DECL FDAT FP87={TOOL_NO 1,BASE_NO 0,IPO_FRAME #BASE,POINT2[] " ",TQ_STATE FALSE}
DECL PDAT PPDAT66={ACC 100.000,APO_DIST 100.000,APO_MODE #CPTP,GEAR_JERK 50.0000}
DECL E6POS XP87={X 1397.26331,Y -207.500198,Z 1611.62207,A -136.868607,B 85.8667068,C -39.2035751,S 2,T 2,E1 229.997360,E2 195.002197,E3 195.004211,E4 0.0,E5 0.0,E6 0.0}
DECL ATBg_Crater_T AC_WDAT46={JobModeId -187662529,ParamSetId -1375177600,CraterTime 0.100000,PostflowTime 0.100000,Channel1 30.0000,Channel2 1.00000,Channel3 0.0,Channel4 0.0,Channel5 0.0,Channel6 0.0,Channel7 0.0,Channel8 0.0,BurnBackTime 0.0}
DECL FDAT FP88={TOOL_NO 1,BASE_NO 0,IPO_FRAME #BASE,POINT2[] " ",TQ_STATE FALSE}
DECL LDAT LCPDAT25={ACC 100.000,APO_DIST 100.000,APO_FAC 50.0000,AXIS_VEL 100.000,AXIS_ACC 100.000,ORI_TYP #VAR,CIRC_TYP #BASE,JERK_FAC 50.0000,GEAR_JERK 50.0000,EXAX_IGN 0}
DECL E6POS XP88={X 1397.26331,Y -207.500198,Z 1611.62207,A -136.868607,B 85.8667068,C -39.2035751,S 2,T 2,E1 229.997360,E2 195.002197,E3 195.004211,E4 0.0,E5 0.0,E6 0.0}
DECL E6POS XP89={X 1306.19275,Y -196.588913,Z 1703.97925,A -68.7830734,B 86.4150162,C 29.0020599,S 2,T 2,E1 229.997360,E2 195.002197,E3 195.004211,E4 0.0,E5 0.0,E6 0.0}
DECL FDAT FP89={TOOL_NO 1,BASE_NO 0,IPO_FRAME #BASE,POINT2[] " ",TQ_STATE FALSE}
DECL PDAT PPDAT67={VEL 100.000,ACC 100.000,APO_DIST 100.000,APO_MODE #CDIS,GEAR_JERK 50.0000,EXAX_IGN 3}
DECL ATBg_Start_T AS_WDAT47={JobModeId -187662529,ParamSetId 687014726,StartTime 0.0,PreFlowTime 0.100000,Channel1 30.0000,Channel2 1.00000,Channel3 0.0,Channel4 0.0,Channel5 0.0,Channel6 0.0,Channel7 0.0,Channel8 0.0,PurgeTime 0.0}
DECL ATBg_Weld_T AW_WDAT47={JobModeId -187662529,ParamSetId -430485013,Velocity 0.00830000,Channel1 30.0000,Channel2 1.00000,Channel3 0.0,Channel4 0.0,Channel5 0.0,Channel6 0.0,Channel7 0.0,Channel8 0.0}
DECL WTCg_WeaveDefinition_T WV_WDAT47={Pattern #None,Length 4.00000,Amplitude 2.00000,Angle 0.0}
DECL FDAT FP90={TOOL_NO 1,BASE_NO 0,IPO_FRAME #BASE,POINT2[] " ",TQ_STATE FALSE}
DECL PDAT PPDAT68={ACC 100.000,APO_DIST 100.000,APO_MODE #CPTP,GEAR_JERK 50.0000}
DECL E6POS XP90={X 1232.65955,Y -891.276917,Z 1635.28589,A -96.7124100,B 54.7162971,C 6.76454,S 2,T 10,E1 229.997360,E2 195.002197,E3 195.004211,E4 0.0,E5 0.0,E6 0.0}
DECL ATBg_Crater_T AC_WDAT48={JobModeId -187662529,ParamSetId -1375177600,CraterTime 0.100000,PostflowTime 0.100000,Channel1 30.0000,Channel2 1.00000,Channel3 0.0,Channel4 0.0,Channel5 0.0,Channel6 0.0,Channel7 0.0,Channel8 0.0,BurnBackTime 0.0}
DECL FDAT FP91={TOOL_NO 1,BASE_NO 0,IPO_FRAME #BASE,POINT2[] " ",TQ_STATE FALSE}
DECL LDAT LCPDAT26={ACC 100.000,APO_DIST 100.000,APO_FAC 50.0000,AXIS_VEL 100.000,AXIS_ACC 100.000,ORI_TYP #VAR,CIRC_TYP #BASE,JERK_FAC 50.0000,GEAR_JERK 50.0000,EXAX_IGN 0}
DECL E6POS XP91={X 1232.65955,Y -891.276917,Z 1635.28589,A -96.7124100,B 54.7162971,C 6.76454,S 2,T 10,E1 229.997360,E2 195.002197,E3 195.004211,E4 0.0,E5 0.0,E6 0.0}
DECL E6POS XP92={X 1054.34692,Y -757.859863,Z 1864.28418,A -84.9267426,B 47.8384056,C 21.8099632,S 2,T 10,E1 229.997360,E2 195.002197,E3 195.004211,E4 0.0,E5 0.0,E6 0.0}
DECL FDAT FP92={TOOL_NO 1,BASE_NO 0,IPO_FRAME #BASE,POINT2[] " ",TQ_STATE FALSE}
DECL PDAT PPDAT69={VEL 100.000,ACC 100.000,APO_DIST 100.000,APO_MODE #CDIS,GEAR_JERK 50.0000,EXAX_IGN 3}
DECL E6POS XP93={X 1192.32471,Y 472.459,Z 1776.73877,A 83.1334229,B 67.4761200,C 156.576218,S 2,T 35,E1 229.997406,E2 195.002228,E3 195.004227,E4 0.0,E5 0.0,E6 0.0}
DECL FDAT FP93={TOOL_NO 1,BASE_NO 0,IPO_FRAME #BASE,POINT2[] " ",TQ_STATE FALSE}
DECL PDAT PPDAT70={VEL 100.000,ACC 100.000,APO_DIST 100.000,APO_MODE #CDIS,GEAR_JERK 50.0000,EXAX_IGN 3}
DECL E6POS XP94={X 1203.56567,Y 245.655396,Z 1802.88013,A 72.3533630,B 68.4953918,C 154.352661,S 2,T 35,E1 229.997391,E2 195.002228,E3 195.004227,E4 0.0,E5 0.0,E6 0.0}
DECL FDAT FP94={TOOL_NO 1,BASE_NO 0,IPO_FRAME #BASE,POINT2[] " ",TQ_STATE FALSE}
DECL PDAT PPDAT71={VEL 100.000,ACC 100.000,APO_DIST 100.000,APO_MODE #CDIS,GEAR_JERK 50.0000,EXAX_IGN 3}
DECL E6POS XP95={X 1366.39880,Y 202.321213,Z 1652.72510,A 92.5657654,B 80.7616730,C 174.120758,S 2,T 35,E1 229.997360,E2 195.002197,E3 195.004211,E4 0.0,E5 0.0,E6 0.0}
DECL FDAT FP95={TOOL_NO 1,BASE_NO 0,IPO_FRAME #BASE,POINT2[] " ",TQ_STATE FALSE}
DECL PDAT PPDAT72={VEL 100.000,ACC 100.000,APO_DIST 100.000,APO_MODE #CDIS,GEAR_JERK 50.0000,EXAX_IGN 3}
DECL E6POS XP96={X 1171.60815,Y -889.236572,Z 1696.34497,A -96.0087738,B 50.3284950,C 9.56970692,S 2,T 10,E1 190.873,E2 195.002197,E3 195.004211,E4 0.0,E5 0.0,E6 0.0}
DECL FDAT FP96={TOOL_NO 1,BASE_NO 0,IPO_FRAME #BASE,POINT2[] " ",TQ_STATE FALSE}
DECL PDAT PPDAT73={VEL 100.000,ACC 100.000,APO_DIST 100.000,APO_MODE #CDIS,GEAR_JERK 50.0000,EXAX_IGN 3}
DECL ATBg_Start_T AS_WDAT49={JobModeId -187662529,ParamSetId 687014726,StartTime 0.0,PreFlowTime 0.100000,Channel1 30.0000,Channel2 1.00000,Channel3 0.0,Channel4 0.0,Channel5 0.0,Channel6 0.0,Channel7 0.0,Channel8 0.0,PurgeTime 0.0}
DECL ATBg_Weld_T AW_WDAT49={JobModeId -187662529,ParamSetId -430485013,Velocity 0.00830000,Channel1 30.0000,Channel2 1.00000,Channel3 0.0,Channel4 0.0,Channel5 0.0,Channel6 0.0,Channel7 0.0,Channel8 0.0}
DECL WTCg_WeaveDefinition_T WV_WDAT49={Pattern #None,Length 4.00000,Amplitude 2.00000,Angle 0.0}
DECL FDAT FP97={TOOL_NO 1,BASE_NO 0,IPO_FRAME #BASE,POINT2[] " ",TQ_STATE FALSE}
DECL PDAT PPDAT74={ACC 100.000,APO_DIST 100.000,APO_MODE #CPTP,GEAR_JERK 50.0000}
DECL E6POS XP97={X 1206.43689,Y -921.566711,Z 1635.16187,A -94.9919662,B 61.2246590,C 10.2442360,S 2,T 10,E1 190.873,E2 195.002197,E3 195.004211,E4 0.0,E5 0.0,E6 0.0}
DECL ATBg_Crater_T AC_WDAT50={JobModeId -187662529,ParamSetId -1375177600,CraterTime 0.100000,PostflowTime 0.100000,Channel1 30.0000,Channel2 1.00000,Channel3 0.0,Channel4 0.0,Channel5 0.0,Channel6 0.0,Channel7 0.0,Channel8 0.0,BurnBackTime 0.0}
DECL FDAT FP98={TOOL_NO 1,BASE_NO 0,IPO_FRAME #BASE,POINT2[] " ",TQ_STATE FALSE}
DECL LDAT LCPDAT27={ACC 100.000,APO_DIST 100.000,APO_FAC 50.0000,AXIS_VEL 100.000,AXIS_ACC 100.000,ORI_TYP #VAR,CIRC_TYP #BASE,JERK_FAC 50.0000,GEAR_JERK 50.0000,EXAX_IGN 0}
DECL E6POS XP98={X 1206.43689,Y -921.566711,Z 1635.16187,A -94.9919662,B 61.2246590,C 10.2442360,S 2,T 10,E1 190.873,E2 195.002197,E3 195.004211,E4 0.0,E5 0.0,E6 0.0}
DECL ATBg_Crater_T AC_WDAT51={JobModeId -187662529,ParamSetId -1375177600,CraterTime 0.100000,PostflowTime 0.100000,Channel1 30.0000,Channel2 1.00000,Channel3 0.0,Channel4 0.0,Channel5 0.0,Channel6 0.0,Channel7 0.0,Channel8 0.0,BurnBackTime 0.0}
DECL FDAT FP99={TOOL_NO 1,BASE_NO 0,IPO_FRAME #BASE,POINT2[] " ",TQ_STATE FALSE}
DECL LDAT LCPDAT28={ACC 100.000,APO_DIST 100.000,APO_FAC 50.0000,AXIS_VEL 100.000,AXIS_ACC 100.000,ORI_TYP #VAR,CIRC_TYP #BASE,JERK_FAC 50.0000,GEAR_JERK 50.0000,EXAX_IGN 0}
DECL E6POS XP99={X 1194.17407,Y -927.370056,Z 1636.72192,A -96.0782471,B 61.4487839,C 9.53255939,S 2,T 10,E1 190.873,E2 195.002197,E3 195.004211,E4 0.0,E5 0.0,E6 0.0}
DECL ATBg_Start_T AS_WDAT52={JobModeId -187662529,ParamSetId 687014726,StartTime 0.0,PreFlowTime 0.100000,Channel1 30.0000,Channel2 1.00000,Channel3 0.0,Channel4 0.0,Channel5 0.0,Channel6 0.0,Channel7 0.0,Channel8 0.0,PurgeTime 0.0}
DECL ATBg_Weld_T AW_WDAT52={JobModeId -187662529,ParamSetId -430485013,Velocity 0.00830000,Channel1 30.0000,Channel2 1.00000,Channel3 0.0,Channel4 0.0,Channel5 0.0,Channel6 0.0,Channel7 0.0,Channel8 0.0}
DECL WTCg_WeaveDefinition_T WV_WDAT52={Pattern #None,Length 4.00000,Amplitude 2.00000,Angle 0.0}
DECL FDAT FP100={TOOL_NO 1,BASE_NO 0,IPO_FRAME #BASE,POINT2[] " ",TQ_STATE FALSE}
DECL PDAT PPDAT75={ACC 100.000,APO_DIST 100.000,APO_MODE #CPTP,GEAR_JERK 50.0000}
DECL E6POS XP100={X 1254.47900,Y -806.532104,Z 1613.77075,A -96.0353394,B 70.1869659,C 2.27105737,S 2,T 10,E1 190.873,E2 195.002197,E3 195.004211,E4 0.0,E5 0.0,E6 0.0}
DECL ATBg_Crater_T AC_WDAT53={JobModeId -187662529,ParamSetId -1375177600,CraterTime 0.100000,PostflowTime 0.100000,Channel1 30.0000,Channel2 1.00000,Channel3 0.0,Channel4 0.0,Channel5 0.0,Channel6 0.0,Channel7 0.0,Channel8 0.0,BurnBackTime 0.0}
DECL FDAT FP101={TOOL_NO 1,BASE_NO 0,IPO_FRAME #BASE,POINT2[] " ",TQ_STATE FALSE}
DECL LDAT LCPDAT29={ACC 100.000,APO_DIST 100.000,APO_FAC 50.0000,AXIS_VEL 100.000,AXIS_ACC 100.000,ORI_TYP #VAR,CIRC_TYP #BASE,JERK_FAC 50.0000,GEAR_JERK 50.0000,EXAX_IGN 0}
DECL E6POS XP101={X 1253.55212,Y -812.493896,Z 1618.97900,A -96.4830627,B 65.4992599,C 1.85604811,S 2,T 10,E1 190.873,E2 195.002197,E3 195.004211,E4 0.0,E5 0.0,E6 0.0}
DECL ATBg_Start_T AS_WDAT54={JobModeId -187662529,ParamSetId 687014726,StartTime 0.0,PreFlowTime 0.100000,Channel1 30.0000,Channel2 1.00000,Channel3 0.0,Channel4 0.0,Channel5 0.0,Channel6 0.0,Channel7 0.0,Channel8 0.0,PurgeTime 0.0}
DECL ATBg_Weld_T AW_WDAT54={JobModeId -187662529,ParamSetId -430485013,Velocity 0.00830000,Channel1 30.0000,Channel2 1.00000,Channel3 0.0,Channel4 0.0,Channel5 0.0,Channel6 0.0,Channel7 0.0,Channel8 0.0}
DECL WTCg_WeaveDefinition_T WV_WDAT54={Pattern #None,Length 4.00000,Amplitude 2.00000,Angle 0.0}
DECL FDAT FP102={TOOL_NO 1,BASE_NO 0,IPO_FRAME #BASE,POINT2[] " ",TQ_STATE FALSE}
DECL PDAT PPDAT76={ACC 100.000,APO_DIST 100.000,APO_MODE #CPTP,GEAR_JERK 50.0000}
DECL E6POS XP102={X 1246.51099,Y -824.909851,Z 1637.50818,A -96.9019775,B 54.7476616,C 1.71330380,S 2,T 10,E1 190.873,E2 195.002197,E3 195.004211,E4 0.0,E5 0.0,E6 0.0}
DECL ATBg_Crater_T AC_WDAT55={JobModeId -187662529,ParamSetId -1375177600,CraterTime 0.100000,PostflowTime 0.100000,Channel1 30.0000,Channel2 1.00000,Channel3 0.0,Channel4 0.0,Channel5 0.0,Channel6 0.0,Channel7 0.0,Channel8 0.0,BurnBackTime 0.0}
DECL FDAT FP103={TOOL_NO 1,BASE_NO 0,IPO_FRAME #BASE,POINT2[] " ",TQ_STATE FALSE}
DECL LDAT LCPDAT30={ACC 100.000,APO_DIST 100.000,APO_FAC 50.0000,AXIS_VEL 100.000,AXIS_ACC 100.000,ORI_TYP #VAR,CIRC_TYP #BASE,JERK_FAC 50.0000,GEAR_JERK 50.0000,EXAX_IGN 0}
DECL E6POS XP103={X 1245.91785,Y -828.361267,Z 1642.64575,A -97.0760269,B 51.0904427,C 1.57438397,S 2,T 10,E1 190.873,E2 195.002197,E3 195.004211,E4 0.0,E5 0.0,E6 0.0}
DECL E6POS XP104={X 993.488,Y -653.571472,Z 1941.27576,A -82.8141479,B 41.6257553,C 21.1250896,S 2,T 10,E1 190.873,E2 195.002197,E3 195.004211,E4 0.0,E5 0.0,E6 0.0}
DECL FDAT FP104={TOOL_NO 1,BASE_NO 0,IPO_FRAME #BASE,POINT2[] " ",TQ_STATE FALSE}
DECL PDAT PPDAT77={VEL 100.000,ACC 100.000,APO_DIST 100.000,APO_MODE #CDIS,GEAR_JERK 50.0000,EXAX_IGN 3}
DECL ATBg_Start_T AS_WDAT56={JobModeId -187662529,ParamSetId 687014726,StartTime 0.0,PreFlowTime 0.100000,Channel1 30.0000,Channel2 1.00000,Channel3 0.0,Channel4 0.0,Channel5 0.0,Channel6 0.0,Channel7 0.0,Channel8 0.0,PurgeTime 0.0}
DECL ATBg_Weld_T AW_WDAT56={JobModeId -187662529,ParamSetId -430485013,Velocity 0.00830000,Channel1 30.0000,Channel2 1.00000,Channel3 0.0,Channel4 0.0,Channel5 0.0,Channel6 0.0,Channel7 0.0,Channel8 0.0}
DECL WTCg_WeaveDefinition_T WV_WDAT56={Pattern #None,Length 4.00000,Amplitude 2.00000,Angle 0.0}
DECL FDAT FP105={TOOL_NO 1,BASE_NO 0,IPO_FRAME #BASE,POINT2[] " ",TQ_STATE FALSE}
DECL PDAT PPDAT78={ACC 100.000,APO_DIST 100.000,APO_MODE #CPTP,GEAR_JERK 50.0000}
DECL E6POS XP105={X 1288.91138,Y -655.583923,Z 1673.83777,A -92.6688843,B 61.3095779,C 22.6213436,S 2,T 10,E1 190.873,E2 195.002197,E3 195.004211,E4 0.0,E5 0.0,E6 0.0}
DECL ATBg_Crater_T AC_WDAT57={JobModeId -187662529,ParamSetId -1375177600,CraterTime 0.100000,PostflowTime 0.100000,Channel1 30.0000,Channel2 1.00000,Channel3 0.0,Channel4 0.0,Channel5 0.0,Channel6 0.0,Channel7 0.0,Channel8 0.0,BurnBackTime 0.0}
DECL FDAT FP106={TOOL_NO 1,BASE_NO 0,IPO_FRAME #BASE,POINT2[] " ",TQ_STATE FALSE}
DECL LDAT LCPDAT31={ACC 100.000,APO_DIST 100.000,APO_FAC 50.0000,AXIS_VEL 100.000,AXIS_ACC 100.000,ORI_TYP #VAR,CIRC_TYP #BASE,JERK_FAC 50.0000,GEAR_JERK 50.0000,EXAX_IGN 0}
DECL E6POS XP106={X 1291.79114,Y -651.086548,Z 1668.95923,A -88.7677460,B 65.1891708,C 26.1072254,S 2,T 10,E1 190.873,E2 195.002197,E3 195.004211,E4 0.0,E5 0.0,E6 0.0}
DECL ATBg_Start_T AS_WDAT58={JobModeId -187662529,ParamSetId 687014726,StartTime 0.0,PreFlowTime 0.100000,Channel1 30.0000,Channel2 1.00000,Channel3 0.0,Channel4 0.0,Channel5 0.0,Channel6 0.0,Channel7 0.0,Channel8 0.0,PurgeTime 0.0}
DECL ATBg_Weld_T AW_WDAT58={JobModeId -187662529,ParamSetId -430485013,Velocity 0.00830000,Channel1 30.0000,Channel2 1.00000,Channel3 0.0,Channel4 0.0,Channel5 0.0,Channel6 0.0,Channel7 0.0,Channel8 0.0}
DECL WTCg_WeaveDefinition_T WV_WDAT58={Pattern #None,Length 4.00000,Amplitude 2.00000,Angle 0.0}
DECL FDAT FP107={TOOL_NO 1,BASE_NO 0,IPO_FRAME #BASE,POINT2[] " ",TQ_STATE FALSE}
DECL PDAT PPDAT79={ACC 100.000,APO_DIST 100.000,APO_MODE #CPTP,GEAR_JERK 50.0000}
DECL E6POS XP107={X 1293.96118,Y -629.543518,Z 1661.28882,A -62.0844460,B 76.3225,C 51.4223785,S 2,T 10,E1 190.873,E2 195.002197,E3 195.004211,E4 0.0,E5 0.0,E6 0.0}
DECL ATBg_Crater_T AC_WDAT59={JobModeId -187662529,ParamSetId -1375177600,CraterTime 0.100000,PostflowTime 0.100000,Channel1 30.0000,Channel2 1.00000,Channel3 0.0,Channel4 0.0,Channel5 0.0,Channel6 0.0,Channel7 0.0,Channel8 0.0,BurnBackTime 0.0}
DECL FDAT FP108={TOOL_NO 1,BASE_NO 0,IPO_FRAME #BASE,POINT2[] " ",TQ_STATE FALSE}
DECL LDAT LCPDAT32={ACC 100.000,APO_DIST 100.000,APO_FAC 50.0000,AXIS_VEL 100.000,AXIS_ACC 100.000,ORI_TYP #VAR,CIRC_TYP #BASE,JERK_FAC 50.0000,GEAR_JERK 50.0000,EXAX_IGN 0}
DECL E6POS XP108={X 1296.53784,Y -620.323242,Z 1661.69067,A -61.8037186,B 76.3528748,C 51.3231,S 2,T 10,E1 190.873,E2 195.002197,E3 195.004211,E4 0.0,E5 0.0,E6 0.0}
DECL ATBg_Start_T AS_WDAT60={JobModeId -187662529,ParamSetId 687014726,StartTime 0.0,PreFlowTime 0.100000,Channel1 30.0000,Channel2 1.00000,Channel3 0.0,Channel4 0.0,Channel5 0.0,Channel6 0.0,Channel7 0.0,Channel8 0.0,PurgeTime 0.0}
DECL ATBg_Weld_T AW_WDAT60={JobModeId -187662529,ParamSetId -430485013,Velocity 0.00830000,Channel1 30.0000,Channel2 1.00000,Channel3 0.0,Channel4 0.0,Channel5 0.0,Channel6 0.0,Channel7 0.0,Channel8 0.0}
DECL WTCg_WeaveDefinition_T WV_WDAT60={Pattern #None,Length 4.00000,Amplitude 2.00000,Angle 0.0}
DECL FDAT FP109={TOOL_NO 1,BASE_NO 0,IPO_FRAME #BASE,POINT2[] " ",TQ_STATE FALSE}
DECL PDAT PPDAT80={ACC 100.000,APO_DIST 100.000,APO_MODE #CPTP,GEAR_JERK 50.0000}
DECL E6POS XP109={X 1326.02588,Y -534.179382,Z 1641.57349,A -22.7906227,B 76.3941956,C 71.2853470,S 2,T 10,E1 190.872955,E2 195.002258,E3 195.004166,E4 0.0,E5 0.0,E6 0.0}
DECL ATBg_Crater_T AC_WDAT61={JobModeId -187662529,ParamSetId -1375177600,CraterTime 0.100000,PostflowTime 0.100000,Channel1 30.0000,Channel2 1.00000,Channel3 0.0,Channel4 0.0,Channel5 0.0,Channel6 0.0,Channel7 0.0,Channel8 0.0,BurnBackTime 0.0}
DECL FDAT FP110={TOOL_NO 1,BASE_NO 0,IPO_FRAME #BASE,POINT2[] " ",TQ_STATE FALSE}
DECL LDAT LCPDAT33={ACC 100.000,APO_DIST 100.000,APO_FAC 50.0000,AXIS_VEL 100.000,AXIS_ACC 100.000,ORI_TYP #VAR,CIRC_TYP #BASE,JERK_FAC 50.0000,GEAR_JERK 50.0000,EXAX_IGN 0}
DECL E6POS XP110={X 1323.19653,Y -542.751892,Z 1647.43872,A -43.1925316,B 73.3963852,C 51.5705795,S 2,T 10,E1 190.872955,E2 195.002258,E3 195.004166,E4 0.0,E5 0.0,E6 0.0}
DECL E6POS XP111={X 1280.34766,Y -555.961731,Z 1683.12561,A -42.7582092,B 71.8603516,C 53.2912,S 2,T 10,E1 190.872955,E2 195.002258,E3 195.004166,E4 0.0,E5 0.0,E6 0.0}
DECL FDAT FP111={TOOL_NO 1,BASE_NO 0,IPO_FRAME #BASE,POINT2[] " ",TQ_STATE FALSE}
DECL PDAT PPDAT81={VEL 100.000,ACC 100.000,APO_DIST 100.000,APO_MODE #CDIS,GEAR_JERK 50.0000,EXAX_IGN 3}
DECL E6POS XP112={X 1215.70911,Y -555.400269,Z 1739.47400,A -50.7764931,B 73.0435410,C 52.7764130,S 2,T 10,E1 190.872971,E2 195.002228,E3 195.004196,E4 0.0,E5 0.0,E6 0.0}
DECL FDAT FP112={TOOL_NO 1,BASE_NO 0,IPO_FRAME #BASE,POINT2[] " ",TQ_STATE FALSE}
DECL PDAT PPDAT82={VEL 100.000,ACC 100.000,APO_DIST 100.000,APO_MODE #CDIS,GEAR_JERK 50.0000,EXAX_IGN 3}
DECL ATBg_Start_T AS_WDAT62={JobModeId -187662529,ParamSetId 687014726,StartTime 0.0,PreFlowTime 0.100000,Channel1 30.0000,Channel2 1.00000,Channel3 0.0,Channel4 0.0,Channel5 0.0,Channel6 0.0,Channel7 0.0,Channel8 0.0,PurgeTime 0.0}
DECL ATBg_Weld_T AW_WDAT62={JobModeId -187662529,ParamSetId -430485013,Velocity 0.00830000,Channel1 30.0000,Channel2 1.00000,Channel3 0.0,Channel4 0.0,Channel5 0.0,Channel6 0.0,Channel7 0.0,Channel8 0.0}
DECL WTCg_WeaveDefinition_T WV_WDAT62={Pattern #None,Length 4.00000,Amplitude 2.00000,Angle 0.0}
DECL FDAT FP113={TOOL_NO 1,BASE_NO 0,IPO_FRAME #BASE,POINT2[] " ",TQ_STATE FALSE}
DECL PDAT PPDAT83={ACC 100.000,APO_DIST 100.000,APO_MODE #CPTP,GEAR_JERK 50.0000}
DECL E6POS XP113={X 1296.56372,Y -770.400757,Z 1543.47070,A 0.142972514,B -35.3954086,C -120.373474,S 0,T 34,E1 162.876816,E2 195.002243,E3 195.004135,E4 0.0,E5 0.0,E6 0.0}
DECL E6POS XP114={X 1032.96,Y -606.570557,Z 1836.64832,A 12.8797731,B -52.1382599,C -138.512726,S 0,T 38,E1 162.876816,E2 195.002243,E3 195.004135,E4 0.0,E5 0.0,E6 0.0}
DECL FDAT FP114={TOOL_NO 1,BASE_NO 0,IPO_FRAME #BASE,POINT2[] " ",TQ_STATE FALSE}
DECL PDAT PPDAT84={VEL 100.000,ACC 100.000,APO_DIST 100.000,APO_MODE #CDIS,GEAR_JERK 50.0000,EXAX_IGN 3}
DECL E6POS XP115={X 983.717468,Y -386.217621,Z 1912.19458,A 54.8041496,B -28.0464611,C -156.126465,S 0,T 42,E1 167.538651,E2 195.002243,E3 195.004135,E4 0.0,E5 0.0,E6 0.0}
DECL FDAT FP115={TOOL_NO 1,BASE_NO 0,IPO_FRAME #BASE,POINT2[] " ",TQ_STATE FALSE}
DECL PDAT PPDAT85={VEL 100.000,ACC 100.000,APO_DIST 100.000,APO_MODE #CDIS,GEAR_JERK 50.0000,EXAX_IGN 3}
DECL E6POS XP116={X 1127.12122,Y -538.175171,Z 1741.28772,A 86.2300110,B 45.5118370,C -178.934204,S 2,T 42,E1 180.834290,E2 195.002258,E3 195.004150,E4 0.0,E5 0.0,E6 0.0}
DECL FDAT FP116={TOOL_NO 1,BASE_NO 0,IPO_FRAME #BASE,POINT2[] " ",TQ_STATE FALSE}
DECL PDAT PPDAT86={VEL 100.000,ACC 100.000,APO_DIST 100.000,APO_MODE #CDIS,GEAR_JERK 50.0000,EXAX_IGN 3}
DECL E6POS XP117={X 1223.14966,Y -576.219177,Z 1689.56824,A 62.8018608,B 70.9648209,C 154.731369,S 2,T 10,E1 186.179565,E2 195.002258,E3 195.004166,E4 0.0,E5 0.0,E6 0.0}
DECL FDAT FP117={TOOL_NO 1,BASE_NO 0,IPO_FRAME #BASE,POINT2[] " ",TQ_STATE FALSE}
DECL PDAT PPDAT87={VEL 100.000,ACC 100.000,APO_DIST 100.000,APO_MODE #CDIS,GEAR_JERK 50.0000,EXAX_IGN 3}
DECL E6POS XP118={X 1019.43097,Y -480.945862,Z 1982.61938,A -73.3126068,B 40.0338173,C 23.4100742,S 2,T 10,E1 190.873,E2 195.002197,E3 195.004211,E4 0.0,E5 0.0,E6 0.0}
DECL FDAT FP118={TOOL_NO 1,BASE_NO 0,IPO_FRAME #BASE,POINT2[] " ",TQ_STATE FALSE}
DECL PDAT PPDAT88={VEL 100.000,ACC 100.000,APO_DIST 100.000,APO_MODE #CDIS,GEAR_JERK 50.0000,EXAX_IGN 3}
DECL E6POS XP119={X 1185.85767,Y -519.089905,Z 1836.84534,A -82.4992828,B 53.5618,C 21.6134605,S 2,T 10,E1 190.873,E2 195.002197,E3 195.004211,E4 0.0,E5 0.0,E6 0.0}
DECL FDAT FP119={TOOL_NO 1,BASE_NO 0,IPO_FRAME #BASE,POINT2[] " ",TQ_STATE FALSE}
DECL PDAT PPDAT89={VEL 100.000,ACC 100.000,APO_DIST 100.000,APO_MODE #CDIS,GEAR_JERK 50.0000,EXAX_IGN 3}
DECL ATBg_Crater_T AC_WDAT63={JobModeId -187662529,ParamSetId -1375177600,CraterTime 0.100000,PostflowTime 0.100000,Channel1 30.0000,Channel2 1.00000,Channel3 0.0,Channel4 0.0,Channel5 0.0,Channel6 0.0,Channel7 0.0,Channel8 0.0,BurnBackTime 0.0}
DECL FDAT FP120={TOOL_NO 1,BASE_NO 0,IPO_FRAME #BASE,POINT2[] " ",TQ_STATE FALSE}
DECL LDAT LCPDAT34={ACC 100.000,APO_DIST 100.000,APO_FAC 50.0000,AXIS_VEL 100.000,AXIS_ACC 100.000,ORI_TYP #VAR,CIRC_TYP #BASE,JERK_FAC 50.0000,GEAR_JERK 50.0000,EXAX_IGN 0}
DECL E6POS XP120={X 1296.40698,Y -769.839050,Z 1543.91675,A 0.220987946,B -35.3882370,C -120.418251,S 0,T 34,E1 162.887863,E2 195.002243,E3 195.004135,E4 0.0,E5 0.0,E6 0.0}
DECL E6POS XP121={X 1015.08203,Y -595.076965,Z 1861.00537,A 9.26292515,B -48.8289833,C -133.777206,S 0,T 38,E1 162.887863,E2 195.002243,E3 195.004135,E4 0.0,E5 0.0,E6 0.0}
DECL FDAT FP121={TOOL_NO 1,BASE_NO 0,IPO_FRAME #BASE,POINT2[] " ",TQ_STATE FALSE}
DECL PDAT PPDAT90={VEL 100.000,ACC 100.000,APO_DIST 100.000,APO_MODE #CDIS,GEAR_JERK 50.0000,EXAX_IGN 3}
DECL ATBg_Start_T AS_WDAT64={JobModeId -187662529,ParamSetId 687014726,StartTime 0.0,PreFlowTime 0.100000,Channel1 30.0000,Channel2 1.00000,Channel3 0.0,Channel4 0.0,Channel5 0.0,Channel6 0.0,Channel7 0.0,Channel8 0.0,PurgeTime 0.0}
DECL ATBg_Weld_T AW_WDAT64={JobModeId -187662529,ParamSetId -430485013,Velocity 0.00830000,Channel1 30.0000,Channel2 1.00000,Channel3 0.0,Channel4 0.0,Channel5 0.0,Channel6 0.0,Channel7 0.0,Channel8 0.0}
DECL WTCg_WeaveDefinition_T WV_WDAT64={Pattern #None,Length 4.00000,Amplitude 2.00000,Angle 0.0}
DECL FDAT FP122={TOOL_NO 1,BASE_NO 0,IPO_FRAME #BASE,POINT2[] " ",TQ_STATE FALSE}
DECL PDAT PPDAT91={ACC 100.000,APO_DIST 100.000,APO_MODE #CPTP,GEAR_JERK 50.0000}
DECL E6POS XP122={X 1467.58130,Y -240.404205,Z 1528.18201,A -1.93412697,B -32.3756,C -98.3877335,S 2,T 34,E1 162.887863,E2 195.002243,E3 195.004135,E4 0.0,E5 0.0,E6 0.0}
DECL ATBg_Crater_T AC_WDAT65={JobModeId -187662529,ParamSetId -1375177600,CraterTime 0.100000,PostflowTime 0.100000,Channel1 30.0000,Channel2 1.00000,Channel3 0.0,Channel4 0.0,Channel5 0.0,Channel6 0.0,Channel7 0.0,Channel8 0.0,BurnBackTime 0.0}
DECL FDAT FP123={TOOL_NO 1,BASE_NO 0,IPO_FRAME #BASE,POINT2[] " ",TQ_STATE FALSE}
DECL LDAT LCPDAT35={ACC 100.000,APO_DIST 100.000,APO_FAC 50.0000,AXIS_VEL 100.000,AXIS_ACC 100.000,ORI_TYP #VAR,CIRC_TYP #BASE,JERK_FAC 50.0000,GEAR_JERK 50.0000,EXAX_IGN 0}
DECL E6POS XP123={X 1467.58130,Y -240.404205,Z 1528.18201,A -1.93412697,B -32.3756,C -98.3877335,S 2,T 34,E1 162.887863,E2 195.002243,E3 195.004135,E4 0.0,E5 0.0,E6 0.0}
DECL ATBg_Start_T AS_WDAT66={JobModeId -187662529,ParamSetId 687014726,StartTime 0.0,PreFlowTime 0.100000,Channel1 30.0000,Channel2 1.00000,Channel3 0.0,Channel4 0.0,Channel5 0.0,Channel6 0.0,Channel7 0.0,Channel8 0.0,PurgeTime 0.0}
DECL ATBg_Weld_T AW_WDAT66={JobModeId -187662529,ParamSetId -430485013,Velocity 0.00830000,Channel1 30.0000,Channel2 1.00000,Channel3 0.0,Channel4 0.0,Channel5 0.0,Channel6 0.0,Channel7 0.0,Channel8 0.0}
DECL WTCg_WeaveDefinition_T WV_WDAT66={Pattern #None,Length 4.00000,Amplitude 2.00000,Angle 0.0}
DECL FDAT FP124={TOOL_NO 1,BASE_NO 0,IPO_FRAME #BASE,POINT2[] " ",TQ_STATE FALSE}
DECL PDAT PPDAT92={ACC 100.000,APO_DIST 100.000,APO_MODE #CPTP,GEAR_JERK 50.0000}
DECL E6POS XP124={X 1481.05737,Y 10.8651133,Z 1536.92859,A -3.71409750,B -32.3918381,C -85.6522675,S 2,T 42,E1 162.887863,E2 195.002243,E3 195.004135,E4 0.0,E5 0.0,E6 0.0}
DECL ATBg_Crater_T AC_WDAT67={JobModeId -187662529,ParamSetId -1375177600,CraterTime 0.100000,PostflowTime 0.100000,Channel1 30.0000,Channel2 1.00000,Channel3 0.0,Channel4 0.0,Channel5 0.0,Channel6 0.0,Channel7 0.0,Channel8 0.0,BurnBackTime 0.0}
DECL FDAT FP125={TOOL_NO 1,BASE_NO 0,IPO_FRAME #BASE,POINT2[] " ",TQ_STATE FALSE}
DECL LDAT LCPDAT36={ACC 100.000,APO_DIST 100.000,APO_FAC 50.0000,AXIS_VEL 100.000,AXIS_ACC 100.000,ORI_TYP #VAR,CIRC_TYP #BASE,JERK_FAC 50.0000,GEAR_JERK 50.0000,EXAX_IGN 0}
DECL E6POS XP125={X 1481.05737,Y 10.8651133,Z 1536.92859,A -3.71409750,B -32.3918381,C -85.6522675,S 2,T 42,E1 162.887863,E2 195.002243,E3 195.004135,E4 0.0,E5 0.0,E6 0.0}
DECL ATBg_Start_T AS_WDAT68={JobModeId -187662529,ParamSetId 687014726,StartTime 0.0,PreFlowTime 0.100000,Channel1 30.0000,Channel2 1.00000,Channel3 0.0,Channel4 0.0,Channel5 0.0,Channel6 0.0,Channel7 0.0,Channel8 0.0,PurgeTime 0.0}
DECL ATBg_Weld_T AW_WDAT68={JobModeId -187662529,ParamSetId -430485013,Velocity 0.00830000,Channel1 30.0000,Channel2 1.00000,Channel3 0.0,Channel4 0.0,Channel5 0.0,Channel6 0.0,Channel7 0.0,Channel8 0.0}
DECL WTCg_WeaveDefinition_T WV_WDAT68={Pattern #None,Length 4.00000,Amplitude 2.00000,Angle 0.0}
DECL FDAT FP126={TOOL_NO 1,BASE_NO 0,IPO_FRAME #BASE,POINT2[] " ",TQ_STATE FALSE}
DECL PDAT PPDAT93={ACC 100.000,APO_DIST 100.000,APO_MODE #CPTP,GEAR_JERK 50.0000}
DECL E6POS XP126={X 1444.21252,Y 329.091553,Z 1578.60730,A -4.10677433,B -37.4463387,C -75.4550400,S 2,T 43,E1 162.887848,E2 195.002243,E3 195.004120,E4 0.0,E5 0.0,E6 0.0}
DECL ATBg_Crater_T AC_WDAT69={JobModeId -187662529,ParamSetId -1375177600,CraterTime 0.100000,PostflowTime 0.100000,Channel1 30.0000,Channel2 1.00000,Channel3 0.0,Channel4 0.0,Channel5 0.0,Channel6 0.0,Channel7 0.0,Channel8 0.0,BurnBackTime 0.0}
DECL FDAT FP127={TOOL_NO 1,BASE_NO 0,IPO_FRAME #BASE,POINT2[] " ",TQ_STATE FALSE}
DECL LDAT LCPDAT37={ACC 100.000,APO_DIST 100.000,APO_FAC 50.0000,AXIS_VEL 100.000,AXIS_ACC 100.000,ORI_TYP #VAR,CIRC_TYP #BASE,JERK_FAC 50.0000,GEAR_JERK 50.0000,EXAX_IGN 0}
DECL E6POS XP127={X 1444.21252,Y 329.091553,Z 1578.60730,A -4.10677433,B -37.4463387,C -75.4550400,S 2,T 43,E1 162.887848,E2 195.002243,E3 195.004120,E4 0.0,E5 0.0,E6 0.0}
DECL ATBg_Start_T AS_WDAT70={JobModeId -187662529,ParamSetId 687014726,StartTime 0.0,PreFlowTime 0.100000,Channel1 30.0000,Channel2 1.00000,Channel3 0.0,Channel4 0.0,Channel5 0.0,Channel6 0.0,Channel7 0.0,Channel8 0.0,PurgeTime 0.0}
DECL ATBg_Weld_T AW_WDAT70={JobModeId -187662529,ParamSetId -430485013,Velocity 0.00830000,Channel1 30.0000,Channel2 1.00000,Channel3 0.0,Channel4 0.0,Channel5 0.0,Channel6 0.0,Channel7 0.0,Channel8 0.0}
DECL WTCg_WeaveDefinition_T WV_WDAT70={Pattern #None,Length 4.00000,Amplitude 2.00000,Angle 0.0}
DECL FDAT FP128={TOOL_NO 1,BASE_NO 0,IPO_FRAME #BASE,POINT2[] " ",TQ_STATE FALSE}
DECL PDAT PPDAT94={ACC 100.000,APO_DIST 100.000,APO_MODE #CPTP,GEAR_JERK 50.0000}
DECL E6POS XP128={X 1444.21252,Y 329.091553,Z 1578.60730,A -4.10677433,B -37.4463387,C -75.4550400,S 2,T 43,E1 162.887848,E2 195.002243,E3 195.004120,E4 0.0,E5 0.0,E6 0.0}
DECL ATBg_Crater_T AC_WDAT71={JobModeId -187662529,ParamSetId -1375177600,CraterTime 0.100000,PostflowTime 0.100000,Channel1 30.0000,Channel2 1.00000,Channel3 0.0,Channel4 0.0,Channel5 0.0,Channel6 0.0,Channel7 0.0,Channel8 0.0,BurnBackTime 0.0}
DECL FDAT FP129={TOOL_NO 1,BASE_NO 0,IPO_FRAME #BASE,POINT2[] " ",TQ_STATE FALSE}
DECL LDAT LCPDAT38={ACC 100.000,APO_DIST 100.000,APO_FAC 50.0000,AXIS_VEL 100.000,AXIS_ACC 100.000,ORI_TYP #VAR,CIRC_TYP #BASE,JERK_FAC 50.0000,GEAR_JERK 50.0000,EXAX_IGN 0}
DECL E6POS XP129={X 1444.21252,Y 329.091553,Z 1578.60730,A -4.10677433,B -37.4463387,C -75.4550400,S 2,T 43,E1 162.887848,E2 195.002243,E3 195.004120,E4 0.0,E5 0.0,E6 0.0}
DECL E6POS XP130={X 1106.52942,Y 227.610046,Z 1915.48096,A -12.1633968,B -55.2442207,C -66.5929108,S 2,T 43,E1 162.887848,E2 195.002243,E3 195.004120,E4 0.0,E5 0.0,E6 0.0}
DECL FDAT FP130={TOOL_NO 1,BASE_NO 0,IPO_FRAME #BASE,POINT2[] " ",TQ_STATE FALSE}
DECL PDAT PPDAT95={VEL 100.000,ACC 100.000,APO_DIST 100.000,APO_MODE #CDIS,GEAR_JERK 50.0000,EXAX_IGN 3}
DECL E6POS XP131={X 1047.66113,Y 425.531586,Z 1914.70532,A -17.3199234,B -49.3159409,C -53.3732643,S 2,T 43,E1 162.887848,E2 195.002243,E3 195.004120,E4 0.0,E5 0.0,E6 0.0}
DECL FDAT FP131={TOOL_NO 1,BASE_NO 0,IPO_FRAME #BASE,POINT2[] " ",TQ_STATE FALSE}
DECL PDAT PPDAT96={VEL 100.000,ACC 100.000,APO_DIST 100.000,APO_MODE #CDIS,GEAR_JERK 50.0000,EXAX_IGN 3}
DECL ATBg_Start_T AS_WDAT72={JobModeId -187662529,ParamSetId 687014726,StartTime 0.0,PreFlowTime 0.100000,Channel1 30.0000,Channel2 1.00000,Channel3 0.0,Channel4 0.0,Channel5 0.0,Channel6 0.0,Channel7 0.0,Channel8 0.0,PurgeTime 0.0}
DECL ATBg_Weld_T AW_WDAT72={JobModeId -187662529,ParamSetId -430485013,Velocity 0.00830000,Channel1 30.0000,Channel2 1.00000,Channel3 0.0,Channel4 0.0,Channel5 0.0,Channel6 0.0,Channel7 0.0,Channel8 0.0}
DECL WTCg_WeaveDefinition_T WV_WDAT72={Pattern #None,Length 4.00000,Amplitude 2.00000,Angle 0.0}
DECL FDAT FP132={TOOL_NO 1,BASE_NO 0,IPO_FRAME #BASE,POINT2[] " ",TQ_STATE FALSE}
DECL PDAT PPDAT97={ACC 100.000,APO_DIST 100.000,APO_MODE #CPTP,GEAR_JERK 50.0000}
DECL E6POS XP132={X 1380.53210,Y 589.161865,Z 1585.12817,A -0.785289049,B -38.0413094,C -68.7817764,S 2,T 43,E1 162.887848,E2 195.002243,E3 195.004120,E4 0.0,E5 0.0,E6 0.0}
DECL ATBg_Crater_T AC_WDAT73={JobModeId -187662529,ParamSetId -1375177600,CraterTime 0.100000,PostflowTime 0.100000,Channel1 30.0000,Channel2 1.00000,Channel3 0.0,Channel4 0.0,Channel5 0.0,Channel6 0.0,Channel7 0.0,Channel8 0.0,BurnBackTime 0.0}
DECL FDAT FP133={TOOL_NO 1,BASE_NO 0,IPO_FRAME #BASE,POINT2[] " ",TQ_STATE FALSE}
DECL LDAT LCPDAT39={ACC 100.000,APO_DIST 100.000,APO_FAC 50.0000,AXIS_VEL 100.000,AXIS_ACC 100.000,ORI_TYP #VAR,CIRC_TYP #BASE,JERK_FAC 50.0000,GEAR_JERK 50.0000,EXAX_IGN 0}
DECL E6POS XP133={X 1380.53210,Y 589.161865,Z 1585.12817,A -0.785289049,B -38.0413094,C -68.7817764,S 2,T 43,E1 162.887848,E2 195.002243,E3 195.004120,E4 0.0,E5 0.0,E6 0.0}
DECL ATBg_Start_T AS_WDAT74={JobModeId -187662529,ParamSetId 687014726,StartTime 0.0,PreFlowTime 0.100000,Channel1 30.0000,Channel2 1.00000,Channel3 0.0,Channel4 0.0,Channel5 0.0,Channel6 0.0,Channel7 0.0,Channel8 0.0,PurgeTime 0.0}
DECL ATBg_Weld_T AW_WDAT74={JobModeId -187662529,ParamSetId -430485013,Velocity 0.00830000,Channel1 30.0000,Channel2 1.00000,Channel3 0.0,Channel4 0.0,Channel5 0.0,Channel6 0.0,Channel7 0.0,Channel8 0.0}
DECL WTCg_WeaveDefinition_T WV_WDAT74={Pattern #None,Length 4.00000,Amplitude 2.00000,Angle 0.0}
DECL FDAT FP134={TOOL_NO 1,BASE_NO 0,IPO_FRAME #BASE,POINT2[] " ",TQ_STATE FALSE}
DECL PDAT PPDAT98={ACC 100.000,APO_DIST 100.000,APO_MODE #CPTP,GEAR_JERK 50.0000}
DECL E6POS XP134={X 1324.21606,Y 577.033569,Z 1675.84180,A 33.2802849,B 68.3659897,C 98.0990524,S 2,T 43,E1 193.523224,E2 195.002243,E3 195.004120,E4 0.0,E5 0.0,E6 0.0}
DECL ATBg_Crater_T AC_WDAT75={JobModeId -187662529,ParamSetId -1375177600,CraterTime 0.100000,PostflowTime 0.100000,Channel1 30.0000,Channel2 1.00000,Channel3 0.0,Channel4 0.0,Channel5 0.0,Channel6 0.0,Channel7 0.0,Channel8 0.0,BurnBackTime 0.0}
DECL FDAT FP135={TOOL_NO 1,BASE_NO 0,IPO_FRAME #BASE,POINT2[] " ",TQ_STATE FALSE}
DECL LDAT LCPDAT40={ACC 100.000,APO_DIST 100.000,APO_FAC 50.0000,AXIS_VEL 100.000,AXIS_ACC 100.000,ORI_TYP #VAR,CIRC_TYP #BASE,JERK_FAC 50.0000,GEAR_JERK 50.0000,EXAX_IGN 0}
DECL E6POS XP135={X 1315.22058,Y 580.528381,Z 1674.43982,A 33.6923904,B 68.7131882,C 98.2455063,S 2,T 43,E1 193.523224,E2 195.002243,E3 195.004120,E4 0.0,E5 0.0,E6 0.0}
DECL E6POS XP136={X 877.952393,Y 378.009613,Z 2066.49194,A 29.4934158,B 46.4165955,C 93.3650665,S 2,T 43,E1 66.3312759,E2 195.002243,E3 195.004120,E4 0.0,E5 0.0,E6 0.0}
DECL FDAT FP136={TOOL_NO 1,BASE_NO 0,IPO_FRAME #BASE,POINT2[] " ",TQ_STATE FALSE}
DECL PDAT PPDAT99={VEL 100.000,ACC 100.000,APO_DIST 100.000,APO_MODE #CDIS,GEAR_JERK 50.0000,EXAX_IGN 3}
DECL E6POS XP137={X 930.186890,Y 401.235260,Z 2032.07666,A 29.6696663,B 48.8887520,C 93.6704865,S 2,T 43,E1 117.250534,E2 195.002243,E3 195.004120,E4 0.0,E5 0.0,E6 0.0}
DECL FDAT FP137={TOOL_NO 1,BASE_NO 0,IPO_FRAME #BASE,POINT2[] " ",TQ_STATE FALSE}
DECL PDAT PPDAT100={VEL 100.000,ACC 100.000,APO_DIST 100.000,APO_MODE #CDIS,GEAR_JERK 50.0000,EXAX_IGN 3}
DECL E6POS XP138={X 1118.40247,Y -137.306046,Z 1876.11963,A 29.1699791,B -44.9447441,C -129.111099,S 2,T 34,E1 162.887863,E2 195.002243,E3 195.004135,E4 0.0,E5 0.0,E6 0.0}
DECL FDAT FP138={TOOL_NO 1,BASE_NO 0,IPO_FRAME #BASE,POINT2[] " ",TQ_STATE FALSE}
DECL PDAT PPDAT101={VEL 100.000,ACC 100.000,APO_DIST 100.000,APO_MODE #CDIS,GEAR_JERK 50.0000,EXAX_IGN 3}
DECL E6POS XP139={X 1118.40247,Y -137.306061,Z 1876.11963,A 29.1699696,B -44.9447479,C -129.111099,S 2,T 34,E1 162.887863,E2 195.002243,E3 195.004135,E4 0.0,E5 0.0,E6 0.0}
DECL FDAT FP139={TOOL_NO 1,BASE_NO 0,IPO_FRAME #BASE,POINT2[] " ",TQ_STATE FALSE}
DECL PDAT PPDAT102={VEL 100.000,ACC 100.000,APO_DIST 100.000,APO_MODE #CDIS,GEAR_JERK 50.0000,EXAX_IGN 3}
DECL E6POS XP140={X 1130.15820,Y 68.0121,Z 1887.62683,A 1.93376851,B -54.0676651,C -97.8631592,S 2,T 35,E1 162.887863,E2 195.002243,E3 195.004135,E4 0.0,E5 0.0,E6 0.0}
DECL FDAT FP140={TOOL_NO 1,BASE_NO 0,IPO_FRAME #BASE,POINT2[] " ",TQ_STATE FALSE}
DECL PDAT PPDAT103={VEL 100.000,ACC 100.000,APO_DIST 100.000,APO_MODE #CDIS,GEAR_JERK 50.0000,EXAX_IGN 3}
DECL E6POS XP141={X 1438.32813,Y 17.7426624,Z 1580.02771,A -3.33024645,B -33.9155655,C -86.5758896,S 2,T 42,E1 162.887863,E2 195.002243,E3 195.004135,E4 0.0,E5 0.0,E6 0.0}
DECL FDAT FP141={TOOL_NO 1,BASE_NO 0,IPO_FRAME #BASE,POINT2[] " ",TQ_STATE FALSE}
DECL PDAT PPDAT104={VEL 100.000,ACC 100.000,APO_DIST 100.000,APO_MODE #CDIS,GEAR_JERK 50.0000,EXAX_IGN 3}
DECL E6POS XP142={X 1438.32813,Y 17.7426624,Z 1580.02771,A -3.33024645,B -33.9155655,C -86.5758896,S 2,T 42,E1 162.887863,E2 195.002243,E3 195.004135,E4 0.0,E5 0.0,E6 0.0}
DECL FDAT FP142={TOOL_NO 1,BASE_NO 0,IPO_FRAME #BASE,POINT2[] " ",TQ_STATE FALSE}
DECL PDAT PPDAT105={VEL 100.000,ACC 100.000,APO_DIST 100.000,APO_MODE #CDIS,GEAR_JERK 50.0000,EXAX_IGN 3}
DECL E6POS XP143={X 1343.19556,Y 573.995483,Z 1631.42358,A -1.42052090,B -39.8733025,C -67.7716,S 2,T 43,E1 162.887848,E2 195.002243,E3 195.004120,E4 0.0,E5 0.0,E6 0.0}
DECL FDAT FP143={TOOL_NO 1,BASE_NO 0,IPO_FRAME #BASE,POINT2[] " ",TQ_STATE FALSE}
DECL PDAT PPDAT106={VEL 100.000,ACC 100.000,APO_DIST 100.000,APO_MODE #CDIS,GEAR_JERK 50.0000,EXAX_IGN 3}
DECL E6POS XP144={X 1273.17053,Y 587.464966,Z 1698.79993,A 83.2784653,B 60.5438156,C 145.168457,S 2,T 43,E1 190.194763,E2 195.002243,E3 195.004120,E4 0.0,E5 0.0,E6 0.0}
DECL FDAT FP144={TOOL_NO 1,BASE_NO 0,IPO_FRAME #BASE,POINT2[] " ",TQ_STATE FALSE}
DECL PDAT PPDAT107={VEL 100.000,ACC 100.000,APO_DIST 100.000,APO_MODE #CDIS,GEAR_JERK 50.0000,EXAX_IGN 3}
DECL ATBg_Start_T AS_WDAT76={JobModeId -187662529,ParamSetId 687014726,StartTime 0.0,PreFlowTime 0.100000,Channel1 30.0000,Channel2 1.00000,Channel3 0.0,Channel4 0.0,Channel5 0.0,Channel6 0.0,Channel7 0.0,Channel8 0.0,PurgeTime 0.0}
DECL ATBg_Weld_T AW_WDAT76={JobModeId -187662529,ParamSetId -430485013,Velocity 0.00830000,Channel1 30.0000,Channel2 1.00000,Channel3 0.0,Channel4 0.0,Channel5 0.0,Channel6 0.0,Channel7 0.0,Channel8 0.0}
DECL WTCg_WeaveDefinition_T WV_WDAT76={Pattern #None,Length 4.00000,Amplitude 2.00000,Angle 0.0}
DECL FDAT FP145={TOOL_NO 1,BASE_NO 0,IPO_FRAME #BASE,POINT2[] " ",TQ_STATE FALSE}
DECL PDAT PPDAT108={ACC 100.000,APO_DIST 100.000,APO_MODE #CPTP,GEAR_JERK 50.0000}
DECL E6POS XP145={X 1350.38965,Y 500.946869,Z 1633.47791,A 59.2960243,B 60.0680428,C 137.259659,S 6,T 27,E1 51.7690620,E2 195.002243,E3 195.004120,E4 0.0,E5 0.0,E6 0.0}
DECL ATBg_Crater_T AC_WDAT77={JobModeId -187662529,ParamSetId -1375177600,CraterTime 0.100000,PostflowTime 0.100000,Channel1 30.0000,Channel2 1.00000,Channel3 0.0,Channel4 0.0,Channel5 0.0,Channel6 0.0,Channel7 0.0,Channel8 0.0,BurnBackTime 0.0}
DECL FDAT FP146={TOOL_NO 1,BASE_NO 0,IPO_FRAME #BASE,POINT2[] " ",TQ_STATE FALSE}
DECL LDAT LCPDAT41={ACC 100.000,APO_DIST 100.000,APO_FAC 50.0000,AXIS_VEL 100.000,AXIS_ACC 100.000,ORI_TYP #VAR,CIRC_TYP #BASE,JERK_FAC 50.0000,GEAR_JERK 50.0000,EXAX_IGN 0}
DECL E6POS XP146={X 1350.38965,Y 500.946869,Z 1633.47791,A 59.2960243,B 60.0680428,C 137.259659,S 6,T 27,E1 51.7690620,E2 195.002243,E3 195.004120,E4 0.0,E5 0.0,E6 0.0}
DECL ATBg_Start_T AS_WDAT78={JobModeId -187662529,ParamSetId 687014726,StartTime 0.0,PreFlowTime 0.100000,Channel1 30.0000,Channel2 1.00000,Channel3 0.0,Channel4 0.0,Channel5 0.0,Channel6 0.0,Channel7 0.0,Channel8 0.0,PurgeTime 0.0}
DECL ATBg_Weld_T AW_WDAT78={JobModeId -187662529,ParamSetId -430485013,Velocity 0.00830000,Channel1 30.0000,Channel2 1.00000,Channel3 0.0,Channel4 0.0,Channel5 0.0,Channel6 0.0,Channel7 0.0,Channel8 0.0}
DECL WTCg_WeaveDefinition_T WV_WDAT78={Pattern #None,Length 4.00000,Amplitude 2.00000,Angle 0.0}
DECL FDAT FP147={TOOL_NO 1,BASE_NO 0,IPO_FRAME #BASE,POINT2[] " ",TQ_STATE FALSE}
DECL PDAT PPDAT109={ACC 100.000,APO_DIST 100.000,APO_MODE #CPTP,GEAR_JERK 50.0000}
DECL E6POS XP147={X 1393.22815,Y 126.055344,Z 1638.28113,A 24.8248920,B 64.7499,C 108.646500,S 6,T 27,E1 63.8692,E2 195.002243,E3 195.004120,E4 0.0,E5 0.0,E6 0.0}
DECL ATBg_Start_T AS_WDAT79={JobModeId -187662529,ParamSetId 687014726,StartTime 0.0,PreFlowTime 0.100000,Channel1 30.0000,Channel2 1.00000,Channel3 0.0,Channel4 0.0,Channel5 0.0,Channel6 0.0,Channel7 0.0,Channel8 0.0,PurgeTime 0.0}
DECL ATBg_Weld_T AW_WDAT79={JobModeId -187662529,ParamSetId -430485013,Velocity 0.00830000,Channel1 30.0000,Channel2 1.00000,Channel3 0.0,Channel4 0.0,Channel5 0.0,Channel6 0.0,Channel7 0.0,Channel8 0.0}
DECL WTCg_WeaveDefinition_T WV_WDAT79={Pattern #None,Length 4.00000,Amplitude 2.00000,Angle 0.0}
DECL FDAT FP148={TOOL_NO 1,BASE_NO 0,IPO_FRAME #BASE,POINT2[] " ",TQ_STATE FALSE}
DECL PDAT PPDAT110={ACC 100.000,APO_DIST 100.000,APO_MODE #CPTP,GEAR_JERK 50.0000}
DECL E6POS XP148={X 1391.42883,Y -96.0819855,Z 1637.99084,A 5.40315723,B 62.9757881,C 99.4957809,S 6,T 26,E1 63.8692,E2 195.002243,E3 195.004120,E4 0.0,E5 0.0,E6 0.0}
DECL ATBg_Crater_T AC_WDAT80={JobModeId -187662529,ParamSetId -1375177600,CraterTime 0.100000,PostflowTime 0.100000,Channel1 30.0000,Channel2 1.00000,Channel3 0.0,Channel4 0.0,Channel5 0.0,Channel6 0.0,Channel7 0.0,Channel8 0.0,BurnBackTime 0.0}
DECL FDAT FP149={TOOL_NO 1,BASE_NO 0,IPO_FRAME #BASE,POINT2[] " ",TQ_STATE FALSE}
DECL LDAT LCPDAT42={ACC 100.000,APO_DIST 100.000,APO_FAC 50.0000,AXIS_VEL 100.000,AXIS_ACC 100.000,ORI_TYP #VAR,CIRC_TYP #BASE,JERK_FAC 50.0000,GEAR_JERK 50.0000,EXAX_IGN 0}
DECL E6POS XP149={X 1391.42883,Y -96.0819855,Z 1637.99084,A 5.40315723,B 62.9757881,C 99.4957809,S 6,T 26,E1 63.8692,E2 195.002243,E3 195.004120,E4 0.0,E5 0.0,E6 0.0}
DECL ATBg_Start_T AS_WDAT81={JobModeId -187662529,ParamSetId 687014726,StartTime 0.0,PreFlowTime 0.100000,Channel1 30.0000,Channel2 1.00000,Channel3 0.0,Channel4 0.0,Channel5 0.0,Channel6 0.0,Channel7 0.0,Channel8 0.0,PurgeTime 0.0}
DECL ATBg_Weld_T AW_WDAT81={JobModeId -187662529,ParamSetId -430485013,Velocity 0.00830000,Channel1 30.0000,Channel2 1.00000,Channel3 0.0,Channel4 0.0,Channel5 0.0,Channel6 0.0,Channel7 0.0,Channel8 0.0}
DECL WTCg_WeaveDefinition_T WV_WDAT81={Pattern #None,Length 4.00000,Amplitude 2.00000,Angle 0.0}
DECL FDAT FP150={TOOL_NO 1,BASE_NO 0,IPO_FRAME #BASE,POINT2[] " ",TQ_STATE FALSE}
DECL PDAT PPDAT111={ACC 100.000,APO_DIST 100.000,APO_MODE #CPTP,GEAR_JERK 50.0000}
DECL E6POS XP150={X 1391.42883,Y -96.0819855,Z 1637.99084,A 5.40315723,B 62.9757881,C 99.4957809,S 6,T 26,E1 63.8692,E2 195.002243,E3 195.004120,E4 0.0,E5 0.0,E6 0.0}
DECL ATBg_Crater_T AC_WDAT82={JobModeId -187662529,ParamSetId -1375177600,CraterTime 0.100000,PostflowTime 0.100000,Channel1 30.0000,Channel2 1.00000,Channel3 0.0,Channel4 0.0,Channel5 0.0,Channel6 0.0,Channel7 0.0,Channel8 0.0,BurnBackTime 0.0}
DECL FDAT FP151={TOOL_NO 1,BASE_NO 0,IPO_FRAME #BASE,POINT2[] " ",TQ_STATE FALSE}
DECL LDAT LCPDAT43={ACC 100.000,APO_DIST 100.000,APO_FAC 50.0000,AXIS_VEL 100.000,AXIS_ACC 100.000,ORI_TYP #VAR,CIRC_TYP #BASE,JERK_FAC 50.0000,GEAR_JERK 50.0000,EXAX_IGN 0}
DECL E6POS XP151={X 1391.42883,Y -96.0819855,Z 1637.99084,A 5.40315723,B 62.9757881,C 99.4957809,S 6,T 26,E1 63.8692,E2 195.002243,E3 195.004120,E4 0.0,E5 0.0,E6 0.0}
DECL ATBg_Start_T AS_WDAT83={JobModeId -187662529,ParamSetId 687014726,StartTime 0.0,PreFlowTime 0.100000,Channel1 30.0000,Channel2 1.00000,Channel3 0.0,Channel4 0.0,Channel5 0.0,Channel6 0.0,Channel7 0.0,Channel8 0.0,PurgeTime 0.0}
DECL ATBg_Weld_T AW_WDAT83={JobModeId -187662529,ParamSetId -430485013,Velocity 0.00830000,Channel1 30.0000,Channel2 1.00000,Channel3 0.0,Channel4 0.0,Channel5 0.0,Channel6 0.0,Channel7 0.0,Channel8 0.0}
DECL WTCg_WeaveDefinition_T WV_WDAT83={Pattern #None,Length 4.00000,Amplitude 2.00000,Angle 0.0}
DECL FDAT FP152={TOOL_NO 1,BASE_NO 0,IPO_FRAME #BASE,POINT2[] " ",TQ_STATE FALSE}
DECL PDAT PPDAT112={ACC 100.000,APO_DIST 100.000,APO_MODE #CPTP,GEAR_JERK 50.0000}
DECL E6POS XP152={X 1338.18860,Y -536.074524,Z 1647.32874,A -57.8892822,B 63.7091942,C 41.0981369,S 2,T 10,E1 63.8692,E2 195.002243,E3 195.004120,E4 0.0,E5 0.0,E6 0.0}
DECL ATBg_Crater_T AC_WDAT84={JobModeId -187662529,ParamSetId -1375177600,CraterTime 0.100000,PostflowTime 0.100000,Channel1 30.0000,Channel2 1.00000,Channel3 0.0,Channel4 0.0,Channel5 0.0,Channel6 0.0,Channel7 0.0,Channel8 0.0,BurnBackTime 0.0}
DECL FDAT FP153={TOOL_NO 1,BASE_NO 0,IPO_FRAME #BASE,POINT2[] " ",TQ_STATE FALSE}
DECL LDAT LCPDAT44={ACC 100.000,APO_DIST 100.000,APO_FAC 50.0000,AXIS_VEL 100.000,AXIS_ACC 100.000,ORI_TYP #VAR,CIRC_TYP #BASE,JERK_FAC 50.0000,GEAR_JERK 50.0000,EXAX_IGN 0}
DECL E6POS XP153={X 1338.18860,Y -536.074524,Z 1647.32874,A -57.8892822,B 63.7091942,C 41.0981369,S 2,T 10,E1 63.8692,E2 195.002243,E3 195.004120,E4 0.0,E5 0.0,E6 0.0}
DECL ATBg_Start_T AS_WDAT85={JobModeId -187662529,ParamSetId 687014726,StartTime 0.0,PreFlowTime 0.100000,Channel1 30.0000,Channel2 1.00000,Channel3 0.0,Channel4 0.0,Channel5 0.0,Channel6 0.0,Channel7 0.0,Channel8 0.0,PurgeTime 0.0}
DECL ATBg_Weld_T AW_WDAT85={JobModeId -187662529,ParamSetId -430485013,Velocity 0.00830000,Channel1 30.0000,Channel2 1.00000,Channel3 0.0,Channel4 0.0,Channel5 0.0,Channel6 0.0,Channel7 0.0,Channel8 0.0}
DECL WTCg_WeaveDefinition_T WV_WDAT85={Pattern #None,Length 4.00000,Amplitude 2.00000,Angle 0.0}
DECL FDAT FP154={TOOL_NO 1,BASE_NO 0,IPO_FRAME #BASE,POINT2[] " ",TQ_STATE FALSE}
DECL PDAT PPDAT113={ACC 100.000,APO_DIST 100.000,APO_MODE #CPTP,GEAR_JERK 50.0000}
DECL E6POS XP154={X 1262.58118,Y -864.338440,Z 1614.00354,A -73.6334381,B 51.8891182,C 20.1776752,S 2,T 10,E1 63.8692,E2 195.002243,E3 195.004120,E4 0.0,E5 0.0,E6 0.0}
DECL ATBg_Crater_T AC_WDAT86={JobModeId -187662529,ParamSetId -1375177600,CraterTime 0.100000,PostflowTime 0.100000,Channel1 30.0000,Channel2 1.00000,Channel3 0.0,Channel4 0.0,Channel5 0.0,Channel6 0.0,Channel7 0.0,Channel8 0.0,BurnBackTime 0.0}
DECL FDAT FP155={TOOL_NO 1,BASE_NO 0,IPO_FRAME #BASE,POINT2[] " ",TQ_STATE FALSE}
DECL LDAT LCPDAT45={ACC 100.000,APO_DIST 100.000,APO_FAC 50.0000,AXIS_VEL 100.000,AXIS_ACC 100.000,ORI_TYP #VAR,CIRC_TYP #BASE,JERK_FAC 50.0000,GEAR_JERK 50.0000,EXAX_IGN 0}
DECL E6POS XP155={X 1262.58118,Y -864.338440,Z 1614.00354,A -73.6334381,B 51.8891182,C 20.1776752,S 2,T 10,E1 63.8692,E2 195.002243,E3 195.004120,E4 0.0,E5 0.0,E6 0.0}
DECL E6POS XP156={X 1161.57153,Y -787.106750,Z 1730.94080,A -70.7340851,B 48.4049530,C 23.9520893,S 2,T 10,E1 63.8692,E2 195.002243,E3 195.004120,E4 0.0,E5 0.0,E6 0.0}
DECL FDAT FP156={TOOL_NO 1,BASE_NO 0,IPO_FRAME #BASE,POINT2[] " ",TQ_STATE FALSE}
DECL PDAT PPDAT114={VEL 100.000,ACC 100.000,APO_DIST 100.000,APO_MODE #CDIS,GEAR_JERK 50.0000,EXAX_IGN 3}
DECL E6POS XP157={X 1126.74866,Y 408.069397,Z 1841.40271,A 51.3672,B 51.7329292,C 127.716705,S 6,T 27,E1 51.7690620,E2 195.002243,E3 195.004120,E4 0.0,E5 0.0,E6 0.0}
DECL FDAT FP157={TOOL_NO 1,BASE_NO 0,IPO_FRAME #BASE,POINT2[] " ",TQ_STATE FALSE}
DECL PDAT PPDAT115={VEL 100.000,ACC 100.000,APO_DIST 100.000,APO_MODE #CDIS,GEAR_JERK 50.0000,EXAX_IGN 3}
DECL E6POS XP158={X 1302.66907,Y 210.702881,Z 1692.58154,A 8.67756748,B 64.1599197,C 93.2300949,S 6,T 27,E1 59.8376503,E2 195.002243,E3 195.004120,E4 0.0,E5 0.0,E6 0.0}
DECL FDAT FP158={TOOL_NO 1,BASE_NO 0,IPO_FRAME #BASE,POINT2[] " ",TQ_STATE FALSE}
DECL PDAT PPDAT116={VEL 100.000,ACC 100.000,APO_DIST 100.000,APO_MODE #CDIS,GEAR_JERK 50.0000,EXAX_IGN 3}
DECL E6POS XP159={X 1321.23755,Y 118.253990,Z 1679.97705,A 23.9074345,B 63.3932915,C 107.626610,S 6,T 27,E1 63.8688583,E2 195.002243,E3 195.004120,E4 0.0,E5 0.0,E6 0.0}
DECL FDAT FP159={TOOL_NO 1,BASE_NO 0,IPO_FRAME #BASE,POINT2[] " ",TQ_STATE FALSE}
DECL PDAT PPDAT117={VEL 100.000,ACC 100.000,APO_DIST 100.000,APO_MODE #CDIS,GEAR_JERK 50.0000,EXAX_IGN 3}
DECL ATBg_Crater_T AC_WDAT87={JobModeId -187662529,ParamSetId -1375177600,CraterTime 0.100000,PostflowTime 0.100000,Channel1 30.0000,Channel2 1.00000,Channel3 0.0,Channel4 0.0,Channel5 0.0,Channel6 0.0,Channel7 0.0,Channel8 0.0,BurnBackTime 0.0}
DECL FDAT FP160={TOOL_NO 1,BASE_NO 0,IPO_FRAME #BASE,POINT2[] " ",TQ_STATE FALSE}
DECL LDAT LCPDAT46={ACC 100.000,APO_DIST 100.000,APO_FAC 50.0000,AXIS_VEL 100.000,AXIS_ACC 100.000,ORI_TYP #VAR,CIRC_TYP #BASE,JERK_FAC 50.0000,GEAR_JERK 50.0000,EXAX_IGN 0}
DECL E6POS XP160={X 1393.22815,Y 126.055344,Z 1638.28113,A 24.8248920,B 64.7499,C 108.646500,S 6,T 27,E1 63.8692,E2 195.002243,E3 195.004120,E4 0.0,E5 0.0,E6 0.0}
DECL E6POS XP161={X 1172.91736,Y 102.155952,Z 1791.00903,A 21.1160088,B 58.0485039,C 104.429794,S 6,T 27,E1 63.8692,E2 195.002243,E3 195.004120,E4 0.0,E5 0.0,E6 0.0}
DECL FDAT FP161={TOOL_NO 1,BASE_NO 0,IPO_FRAME #BASE,POINT2[] " ",TQ_STATE FALSE}
DECL PDAT PPDAT118={VEL 100.000,ACC 100.000,APO_DIST 100.000,APO_MODE #CDIS,GEAR_JERK 50.0000,EXAX_IGN 3}
DECL E6POS XP162={X 1319.45740,Y -94.4541702,Z 1687.76807,A 6.00046062,B 61.2865181,C 99.9257813,S 6,T 26,E1 63.8692,E2 195.002243,E3 195.004120,E4 0.0,E5 0.0,E6 0.0}
DECL FDAT FP162={TOOL_NO 1,BASE_NO 0,IPO_FRAME #BASE,POINT2[] " ",TQ_STATE FALSE}
DECL PDAT PPDAT119={VEL 100.000,ACC 100.000,APO_DIST 100.000,APO_MODE #CDIS,GEAR_JERK 50.0000,EXAX_IGN 3}
DECL E6POS XP163={X 1105.24890,Y -83.5208740,Z 1816.11963,A 3.68451500,B 54.5741844,C 97.4914474,S 6,T 26,E1 63.8692,E2 195.002243,E3 195.004120,E4 0.0,E5 0.0,E6 0.0}
DECL FDAT FP163={TOOL_NO 1,BASE_NO 0,IPO_FRAME #BASE,POINT2[] " ",TQ_STATE FALSE}
DECL PDAT PPDAT120={VEL 100.000,ACC 100.000,APO_DIST 100.000,APO_MODE #CDIS,GEAR_JERK 50.0000,EXAX_IGN 3}
DECL E6POS XP164={X 1116.65540,Y -300.466644,Z 1807.37952,A -30.0061340,B 65.1442947,C 72.6307373,S 2,T 10,E1 63.8692,E2 195.002243,E3 195.004120,E4 0.0,E5 0.0,E6 0.0}
DECL FDAT FP164={TOOL_NO 1,BASE_NO 0,IPO_FRAME #BASE,POINT2[] " ",TQ_STATE FALSE}
DECL PDAT PPDAT121={VEL 100.000,ACC 100.000,APO_DIST 100.000,APO_MODE #CDIS,GEAR_JERK 50.0000,EXAX_IGN 3}
DECL E6POS XP165={X 1094.76465,Y -436.932404,Z 1850.25781,A -49.5495834,B 55.7893753,C 50.7237625,S 2,T 10,E1 63.8692,E2 195.002243,E3 195.004120,E4 0.0,E5 0.0,E6 0.0}
DECL FDAT FP165={TOOL_NO 1,BASE_NO 0,IPO_FRAME #BASE,POINT2[] " ",TQ_STATE FALSE}
DECL PDAT PPDAT122={VEL 100.000,ACC 100.000,APO_DIST 100.000,APO_MODE #CDIS,GEAR_JERK 50.0000,EXAX_IGN 3}
DECL E6POS XP166={X 1051.96350,Y -673.004822,Z 1817.49390,A -63.4329147,B 55.2390823,C 44.4735641,S 2,T 10,E1 63.8692,E2 195.002243,E3 195.004120,E4 0.0,E5 0.0,E6 0.0}
DECL FDAT FP166={TOOL_NO 1,BASE_NO 0,IPO_FRAME #BASE,POINT2[] " ",TQ_STATE FALSE}
DECL PDAT PPDAT123={VEL 100.000,ACC 100.000,APO_DIST 100.000,APO_MODE #CDIS,GEAR_JERK 50.0000,EXAX_IGN 3}
DECL ATBg_Start_T AS_WDAT88={JobModeId -187662529,ParamSetId 687014726,StartTime 0.0,PreFlowTime 0.100000,Channel1 30.0000,Channel2 1.00000,Channel3 0.0,Channel4 0.0,Channel5 0.0,Channel6 0.0,Channel7 0.0,Channel8 0.0,PurgeTime 0.0}
DECL ATBg_Weld_T AW_WDAT88={JobModeId -187662529,ParamSetId -430485013,Velocity 0.00830000,Channel1 30.0000,Channel2 1.00000,Channel3 0.0,Channel4 0.0,Channel5 0.0,Channel6 0.0,Channel7 0.0,Channel8 0.0}
DECL WTCg_WeaveDefinition_T WV_WDAT88={Pattern #None,Length 4.00000,Amplitude 2.00000,Angle 0.0}
DECL FDAT FP167={TOOL_NO 1,BASE_NO 0,IPO_FRAME #BASE,POINT2[] " ",TQ_STATE FALSE}
DECL PDAT PPDAT124={ACC 100.000,APO_DIST 100.000,APO_MODE #CPTP,GEAR_JERK 50.0000}
DECL E6POS XP167={X 1345.89380,Y -689.801575,Z 1567.35449,A 4.44710493,B -38.9034271,C -121.049332,S 0,T 34,E1 -15.0944824,E2 195.002243,E3 195.004120,E4 0.0,E5 0.0,E6 0.0}
DECL ATBg_Crater_T AC_WDAT89={JobModeId -187662529,ParamSetId -1375177600,CraterTime 0.100000,PostflowTime 0.100000,Channel1 30.0000,Channel2 1.00000,Channel3 0.0,Channel4 0.0,Channel5 0.0,Channel6 0.0,Channel7 0.0,Channel8 0.0,BurnBackTime 0.0}
DECL FDAT FP168={TOOL_NO 1,BASE_NO 0,IPO_FRAME #BASE,POINT2[] " ",TQ_STATE FALSE}
DECL LDAT LCPDAT47={ACC 100.000,APO_DIST 100.000,APO_FAC 50.0000,AXIS_VEL 100.000,AXIS_ACC 100.000,ORI_TYP #VAR,CIRC_TYP #BASE,JERK_FAC 50.0000,GEAR_JERK 50.0000,EXAX_IGN 0}
DECL E6POS XP168={X 1345.89380,Y -689.801575,Z 1567.35449,A 4.44710493,B -38.9034271,C -121.049332,S 0,T 34,E1 -15.0944824,E2 195.002243,E3 195.004120,E4 0.0,E5 0.0,E6 0.0}
DECL E6POS XP169={X 1115.44019,Y -564.918457,Z 1826.14063,A 11.2815619,B -48.6033707,C -130.884140,S 0,T 34,E1 -15.0944824,E2 195.002243,E3 195.004120,E4 0.0,E5 0.0,E6 0.0}
DECL FDAT FP169={TOOL_NO 1,BASE_NO 0,IPO_FRAME #BASE,POINT2[] " ",TQ_STATE FALSE}
DECL PDAT PPDAT125={VEL 100.000,ACC 100.000,APO_DIST 100.000,APO_MODE #CDIS,GEAR_JERK 50.0000,EXAX_IGN 3}
DECL ATBg_Start_T AS_WDAT90={JobModeId -187662529,ParamSetId 687014726,StartTime 0.0,PreFlowTime 0.100000,Channel1 30.0000,Channel2 1.00000,Channel3 0.0,Channel4 0.0,Channel5 0.0,Channel6 0.0,Channel7 0.0,Channel8 0.0,PurgeTime 0.0}
DECL ATBg_Weld_T AW_WDAT90={JobModeId -187662529,ParamSetId -430485013,Velocity 0.00830000,Channel1 30.0000,Channel2 1.00000,Channel3 0.0,Channel4 0.0,Channel5 0.0,Channel6 0.0,Channel7 0.0,Channel8 0.0}
DECL WTCg_WeaveDefinition_T WV_WDAT90={Pattern #None,Length 4.00000,Amplitude 2.00000,Angle 0.0}
DECL FDAT FP170={TOOL_NO 1,BASE_NO 0,IPO_FRAME #BASE,POINT2[] " ",TQ_STATE FALSE}
DECL PDAT PPDAT126={ACC 100.000,APO_DIST 100.000,APO_MODE #CPTP,GEAR_JERK 50.0000}
DECL E6POS XP170={X 1430.27856,Y -431.329437,Z 1568.64136,A -0.463984519,B -40.1669731,C -106.484306,S 2,T 34,E1 -15.0944824,E2 195.002243,E3 195.004120,E4 0.0,E5 0.0,E6 0.0}
DECL ATBg_Crater_T AC_WDAT91={JobModeId -187662529,ParamSetId -1375177600,CraterTime 0.100000,PostflowTime 0.100000,Channel1 30.0000,Channel2 1.00000,Channel3 0.0,Channel4 0.0,Channel5 0.0,Channel6 0.0,Channel7 0.0,Channel8 0.0,BurnBackTime 0.0}
DECL FDAT FP171={TOOL_NO 1,BASE_NO 0,IPO_FRAME #BASE,POINT2[] " ",TQ_STATE FALSE}
DECL LDAT LCPDAT48={ACC 100.000,APO_DIST 100.000,APO_FAC 50.0000,AXIS_VEL 100.000,AXIS_ACC 100.000,ORI_TYP #VAR,CIRC_TYP #BASE,JERK_FAC 50.0000,GEAR_JERK 50.0000,EXAX_IGN 0}
DECL E6POS XP171={X 1430.27856,Y -431.329437,Z 1568.64136,A -0.463984519,B -40.1669731,C -106.484306,S 2,T 34,E1 -15.0944824,E2 195.002243,E3 195.004120,E4 0.0,E5 0.0,E6 0.0}
DECL E6POS XP172={X 1340.88623,Y -402.247284,Z 1672.75110,A 0.846814,B -44.5353661,C -108.428535,S 2,T 34,E1 -15.0944824,E2 195.002243,E3 195.004120,E4 0.0,E5 0.0,E6 0.0}
DECL FDAT FP172={TOOL_NO 1,BASE_NO 0,IPO_FRAME #BASE,POINT2[] " ",TQ_STATE FALSE}
DECL PDAT PPDAT127={VEL 100.000,ACC 100.000,APO_DIST 100.000,APO_MODE #CDIS,GEAR_JERK 50.0000,EXAX_IGN 3}
DECL E6POS XP173={X 1319.30261,Y -675.391785,Z 1607.84973,A 5.64195442,B -41.0563393,C -122.908539,S 0,T 34,E1 -15.0944824,E2 195.002243,E3 195.004120,E4 0.0,E5 0.0,E6 0.0}
DECL FDAT FP173={TOOL_NO 1,BASE_NO 0,IPO_FRAME #BASE,POINT2[] " ",TQ_STATE FALSE}
DECL PDAT PPDAT128={VEL 100.000,ACC 100.000,APO_DIST 100.000,APO_MODE #CDIS,GEAR_JERK 50.0000,EXAX_IGN 3}
DECL E6POS XP174={X 1340.88623,Y -402.247284,Z 1672.75110,A 0.846814,B -44.5353661,C -108.428535,S 2,T 34,E1 -15.0944824,E2 195.002243,E3 195.004120,E4 0.0,E5 0.0,E6 0.0}
DECL FDAT FP174={TOOL_NO 1,BASE_NO 0,IPO_FRAME #BASE,POINT2[] " ",TQ_STATE FALSE}
DECL PDAT PPDAT129={VEL 100.000,ACC 100.000,APO_DIST 100.000,APO_MODE #CDIS,GEAR_JERK 50.0000,EXAX_IGN 3}
DECL ATBg_Start_T AS_WDAT92={JobModeId -187662529,ParamSetId 687014726,StartTime 0.0,PreFlowTime 0.100000,Channel1 30.0000,Channel2 1.00000,Channel3 0.0,Channel4 0.0,Channel5 0.0,Channel6 0.0,Channel7 0.0,Channel8 0.0,PurgeTime 0.0}
DECL ATBg_Weld_T AW_WDAT92={JobModeId -187662529,ParamSetId -430485013,Velocity 0.00830000,Channel1 30.0000,Channel2 1.00000,Channel3 0.0,Channel4 0.0,Channel5 0.0,Channel6 0.0,Channel7 0.0,Channel8 0.0}
DECL WTCg_WeaveDefinition_T WV_WDAT92={Pattern #None,Length 4.00000,Amplitude 2.00000,Angle 0.0}
DECL FDAT FP175={TOOL_NO 1,BASE_NO 0,IPO_FRAME #BASE,POINT2[] " ",TQ_STATE FALSE}
DECL PDAT PPDAT130={ACC 100.000,APO_DIST 100.000,APO_MODE #CPTP,GEAR_JERK 50.0000}
DECL E6POS XP175={X 1473.60986,Y -91.8296127,Z 1579.61023,A -3.94931197,B -41.4006348,C -87.8952255,S 2,T 42,E1 -15.0945082,E2 195.002151,E3 195.004089,E4 0.0,E5 0.0,E6 0.0}
DECL ATBg_Crater_T AC_WDAT93={JobModeId -187662529,ParamSetId -1375177600,CraterTime 0.100000,PostflowTime 0.100000,Channel1 30.0000,Channel2 1.00000,Channel3 0.0,Channel4 0.0,Channel5 0.0,Channel6 0.0,Channel7 0.0,Channel8 0.0,BurnBackTime 0.0}
DECL FDAT FP176={TOOL_NO 1,BASE_NO 0,IPO_FRAME #BASE,POINT2[] " ",TQ_STATE FALSE}
DECL LDAT LCPDAT49={ACC 100.000,APO_DIST 100.000,APO_FAC 50.0000,AXIS_VEL 100.000,AXIS_ACC 100.000,ORI_TYP #VAR,CIRC_TYP #BASE,JERK_FAC 50.0000,GEAR_JERK 50.0000,EXAX_IGN 0}
DECL E6POS XP176={X 1473.60986,Y -91.8296127,Z 1579.61023,A -3.94931197,B -41.4006348,C -87.8952255,S 2,T 42,E1 -15.0945082,E2 195.002151,E3 195.004089,E4 0.0,E5 0.0,E6 0.0}
DECL ATBg_Start_T AS_WDAT94={JobModeId -187662529,ParamSetId 687014726,StartTime 0.0,PreFlowTime 0.100000,Channel1 30.0000,Channel2 1.00000,Channel3 0.0,Channel4 0.0,Channel5 0.0,Channel6 0.0,Channel7 0.0,Channel8 0.0,PurgeTime 0.0}
DECL ATBg_Weld_T AW_WDAT94={JobModeId -187662529,ParamSetId -430485013,Velocity 0.00830000,Channel1 30.0000,Channel2 1.00000,Channel3 0.0,Channel4 0.0,Channel5 0.0,Channel6 0.0,Channel7 0.0,Channel8 0.0}
DECL WTCg_WeaveDefinition_T WV_WDAT94={Pattern #None,Length 4.00000,Amplitude 2.00000,Angle 0.0}
DECL FDAT FP177={TOOL_NO 1,BASE_NO 0,IPO_FRAME #BASE,POINT2[] " ",TQ_STATE FALSE}
DECL PDAT PPDAT131={ACC 100.000,APO_DIST 100.000,APO_MODE #CPTP,GEAR_JERK 50.0000}
DECL E6POS XP177={X 1467.48669,Y 163.778198,Z 1580.61816,A 7.33355141,B -41.5764198,C -91.4063950,S 2,T 43,E1 -15.0945082,E2 195.002151,E3 195.004089,E4 0.0,E5 0.0,E6 0.0}
DECL ATBg_Crater_T AC_WDAT95={JobModeId -187662529,ParamSetId -1375177600,CraterTime 0.100000,PostflowTime 0.100000,Channel1 30.0000,Channel2 1.00000,Channel3 0.0,Channel4 0.0,Channel5 0.0,Channel6 0.0,Channel7 0.0,Channel8 0.0,BurnBackTime 0.0}
DECL FDAT FP178={TOOL_NO 1,BASE_NO 0,IPO_FRAME #BASE,POINT2[] " ",TQ_STATE FALSE}
DECL LDAT LCPDAT50={ACC 100.000,APO_DIST 100.000,APO_FAC 50.0000,AXIS_VEL 100.000,AXIS_ACC 100.000,ORI_TYP #VAR,CIRC_TYP #BASE,JERK_FAC 50.0000,GEAR_JERK 50.0000,EXAX_IGN 0}
DECL E6POS XP178={X 1467.48669,Y 163.778198,Z 1580.61816,A 7.33355141,B -41.5764198,C -91.4063950,S 2,T 43,E1 -15.0945082,E2 195.002151,E3 195.004089,E4 0.0,E5 0.0,E6 0.0}
DECL E6POS XP179={X 1301.48328,Y 149.157791,Z 1778.32690,A 7.88870478,B -52.9349670,C -92.1586151,S 2,T 43,E1 -15.0945082,E2 195.002151,E3 195.004089,E4 0.0,E5 0.0,E6 0.0}
DECL FDAT FP179={TOOL_NO 1,BASE_NO 0,IPO_FRAME #BASE,POINT2[] " ",TQ_STATE FALSE}
DECL PDAT PPDAT132={VEL 100.000,ACC 100.000,APO_DIST 100.000,APO_MODE #CDIS,GEAR_JERK 50.0000,EXAX_IGN 3}
DECL ATBg_Start_T AS_WDAT96={JobModeId -187662529,ParamSetId 687014726,StartTime 0.0,PreFlowTime 0.100000,Channel1 30.0000,Channel2 1.00000,Channel3 0.0,Channel4 0.0,Channel5 0.0,Channel6 0.0,Channel7 0.0,Channel8 0.0,PurgeTime 0.0}
DECL ATBg_Weld_T AW_WDAT96={JobModeId -187662529,ParamSetId -430485013,Velocity 0.00830000,Channel1 30.0000,Channel2 1.00000,Channel3 0.0,Channel4 0.0,Channel5 0.0,Channel6 0.0,Channel7 0.0,Channel8 0.0}
DECL WTCg_WeaveDefinition_T WV_WDAT96={Pattern #None,Length 4.00000,Amplitude 2.00000,Angle 0.0}
DECL FDAT FP180={TOOL_NO 1,BASE_NO 0,IPO_FRAME #BASE,POINT2[] " ",TQ_STATE FALSE}
DECL PDAT PPDAT133={ACC 100.000,APO_DIST 100.000,APO_MODE #CPTP,GEAR_JERK 50.0000}
DECL E6POS XP180={X 1406.94678,Y 538.867798,Z 1576.37537,A -1.21830094,B -38.4161911,C -71.3365860,S 2,T 43,E1 -15.0945082,E2 195.002151,E3 195.004089,E4 0.0,E5 0.0,E6 0.0}
DECL ATBg_Crater_T AC_WDAT97={JobModeId -187662529,ParamSetId -1375177600,CraterTime 0.100000,PostflowTime 0.100000,Channel1 30.0000,Channel2 1.00000,Channel3 0.0,Channel4 0.0,Channel5 0.0,Channel6 0.0,Channel7 0.0,Channel8 0.0,BurnBackTime 0.0}
DECL FDAT FP181={TOOL_NO 1,BASE_NO 0,IPO_FRAME #BASE,POINT2[] " ",TQ_STATE FALSE}
DECL LDAT LCPDAT51={ACC 100.000,APO_DIST 100.000,APO_FAC 50.0000,AXIS_VEL 100.000,AXIS_ACC 100.000,ORI_TYP #VAR,CIRC_TYP #BASE,JERK_FAC 50.0000,GEAR_JERK 50.0000,EXAX_IGN 0}
DECL E6POS XP181={X 1406.94678,Y 538.867798,Z 1576.37537,A -1.21830094,B -38.4161911,C -71.3365860,S 2,T 43,E1 -15.0945082,E2 195.002151,E3 195.004089,E4 0.0,E5 0.0,E6 0.0}
DECL E6POS XP182={X 1239.22363,Y 477.509247,Z 1777.01758,A -5.46240807,B -48.6917725,C -65.2049179,S 0,T 43,E1 -15.0945082,E2 195.002151,E3 195.004089,E4 0.0,E5 0.0,E6 0.0}
DECL FDAT FP182={TOOL_NO 1,BASE_NO 0,IPO_FRAME #BASE,POINT2[] " ",TQ_STATE FALSE}
DECL PDAT PPDAT134={VEL 100.000,ACC 100.000,APO_DIST 100.000,APO_MODE #CDIS,GEAR_JERK 50.0000,EXAX_IGN 3}
DECL E6POS XP183={X 1239.22363,Y 477.509247,Z 1777.01758,A -5.46240807,B -48.6917725,C -65.2049179,S 0,T 43,E1 -15.0945082,E2 195.002151,E3 195.004089,E4 0.0,E5 0.0,E6 0.0}
DECL FDAT FP183={TOOL_NO 1,BASE_NO 0,IPO_FRAME #BASE,POINT2[] " ",TQ_STATE FALSE}
DECL PDAT PPDAT135={VEL 100.000,ACC 100.000,APO_DIST 100.000,APO_MODE #CDIS,GEAR_JERK 50.0000,EXAX_IGN 3}
DECL E6POS XP184={X 1374.48206,Y 155.586990,Z 1703.80115,A 7.64417267,B -48.7668076,C -91.8435059,S 2,T 43,E1 -15.0945082,E2 195.002151,E3 195.004089,E4 0.0,E5 0.0,E6 0.0}
DECL FDAT FP184={TOOL_NO 1,BASE_NO 0,IPO_FRAME #BASE,POINT2[] " ",TQ_STATE FALSE}
DECL PDAT PPDAT136={VEL 100.000,ACC 100.000,APO_DIST 100.000,APO_MODE #CDIS,GEAR_JERK 50.0000,EXAX_IGN 3}
DECL E6POS XP185={X 1297.61536,Y -75.5030289,Z 1792.50964,A -3.57095265,B -54.1264305,C -88.4031143,S 2,T 42,E1 -15.0945082,E2 195.002151,E3 195.004089,E4 0.0,E5 0.0,E6 0.0}
DECL FDAT FP185={TOOL_NO 1,BASE_NO 0,IPO_FRAME #BASE,POINT2[] " ",TQ_STATE FALSE}
DECL PDAT PPDAT137={VEL 100.000,ACC 100.000,APO_DIST 100.000,APO_MODE #CDIS,GEAR_JERK 50.0000,EXAX_IGN 3}
ENDDAT
